// Mitsubishi GX Works2 project: plc0723   PLC: Q02/Q02H

// global labels: Global1
VAR_GLOBAL
  공급후 AT X0 : BOOL;
  공급전 AT X1 : BOOL;
  드릴상 AT X2 : BOOL;
  드릴하 AT X3 : BOOL;
  송출후 AT X4 : BOOL;
  송출전 AT X5 : BOOL;
  배출후 AT X6 : BOOL;
  배출전 AT X7 : BOOL;
  매거진 AT X8 : BOOL;
  비금속 AT X9 : BOOL;
  금속 AT X0A : BOOL;
  공급전솔 AT Y20 : BOOL;
  공급후솔 AT Y21 : BOOL;
  드릴온 AT Y22 : BOOL;
  송출전솔 AT Y23 : BOOL;
  송출후솔 AT Y24 : BOOL;
  배출전솔 AT Y25 : BOOL;
  배출후솔 AT Y26 : BOOL;
  컨베이어 AT Y27 : BOOL;
  가공드릴 AT Y28 : BOOL;
  적색 AT Y29 : BOOL;
  황색 AT Y2A : BOOL;
  녹색 AT Y2B : BOOL;
  pb1 AT X10 : BOOL;
  pb2 AT X11 : BOOL;
  pb3 AT X12 : BOOL;
  비상정지 AT X13 : BOOL;
  초기화 AT X14 : BOOL;
END_VAR

PROGRAM MAIN
VAR
  테스트동작 : BOOL;
  단일동작 : BOOL;
  연속동작 : BOOL;
  금속탐지 : BOOL;
  송출_전 : BOOL;
  공급_전 : BOOL;
  테스트타이머 : TIMER;
  공급_후 : BOOL;
  가공_하 : BOOL;
  배출_전 : BOOL;
  가공_상 : BOOL;
  배출_후 : BOOL;
  송출_후 : BOOL;
  테스트종료 : BOOL;
  황테 : BOOL;
  녹테 : BOOL;
  공급전진 : BOOL;
  물건없음 : TIMER;
  공급후진 : BOOL;
  타이머1 : TIMER;
  가공드릴온 : BOOL;
  드릴하강 : BOOL;
  타이머2 : TIMER;
  가공드릴오프 : BOOL;
  드릴상승 : BOOL;
  송출전진 : BOOL;
  송출후진 : BOOL;
  컨구동 : BOOL;
  금속판별 : BOOL;
  비금속판별 : BOOL;
  금속타이머 : TIMER;
  배출전진 : BOOL;
  배출후진 : BOOL;
  금종 : BOOL;
  비금속타이머 : TIMER;
  비종 : BOOL;
  동작종료 : BOOL;
  연속종료 : BOOL;
  공급전진2 : BOOL;
  녹색램프 : BOOL;
  황색램프 : BOOL;
  반전 : BOOL;
END_VAR
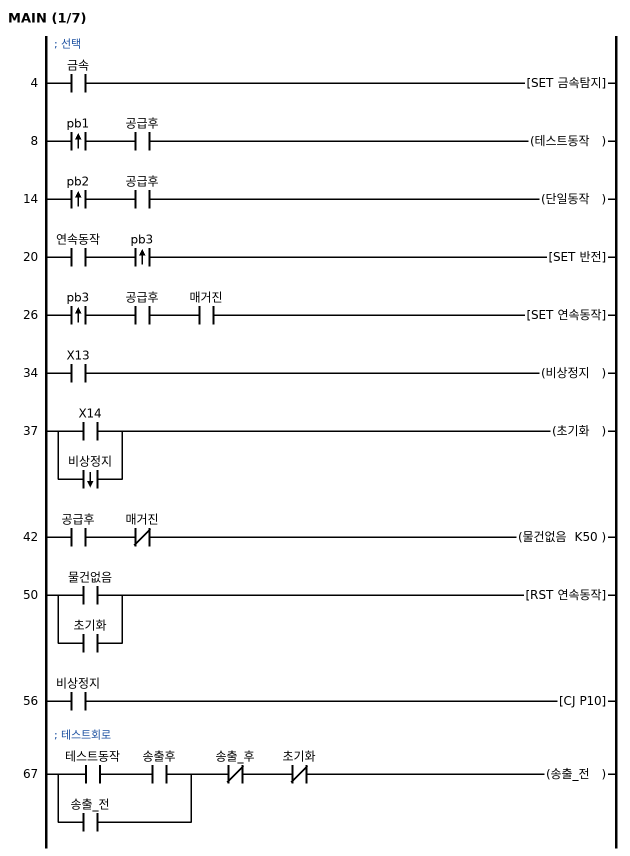
; 선택
4     LD      금속
      SET     금속탐지
8     LDP     pb1
      AND     공급후
      OUT     테스트동작
14    LDP     pb2
      AND     공급후
      OUT     단일동작
20    LD      연속동작
      ANDP    pb3
      SET     반전
26    LDP     pb3
      AND     공급후
      AND     매거진
      SET     연속동작
34    LD      X13
      OUT     비상정지
37    LD      X14
      ORF     비상정지
      OUT     초기화
42    LD      공급후
      ANI     매거진
      OUT     물건없음 K50
50    LD      물건없음
      OR      초기화
      RST     연속동작
56    LD      비상정지
      CJ      P10
; 테스트회로
67    LD      테스트동작
      AND     송출후
      OR      송출_전
      ANI     송출_후
      ANI     초기화
      OUT     송출_전
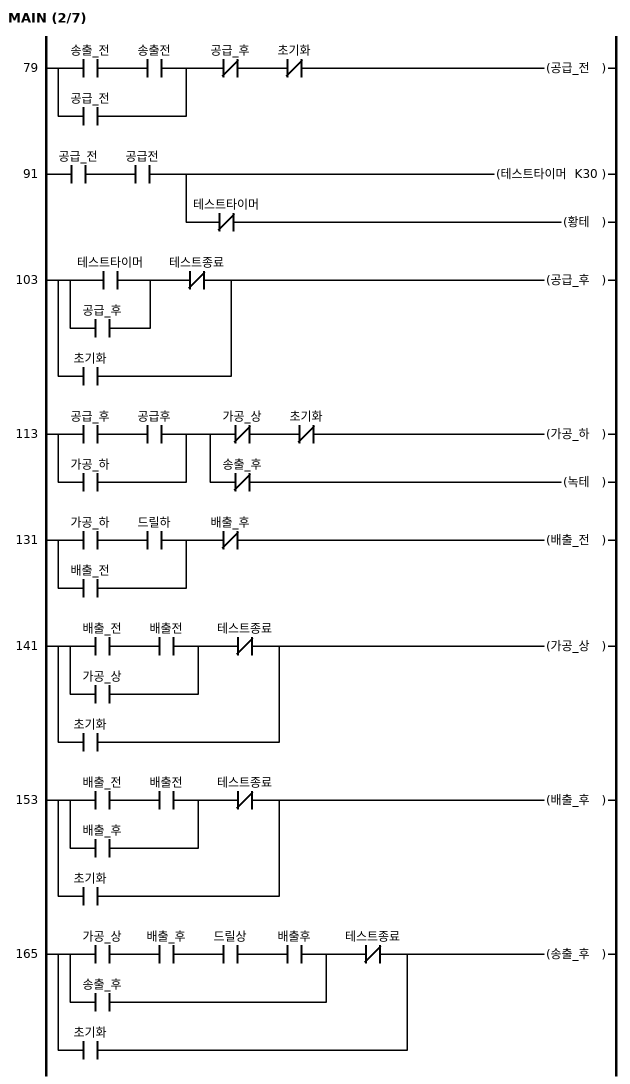
79    LD      송출_전
      AND     송출전
      OR      공급_전
      ANI     공급_후
      ANI     초기화
      OUT     공급_전
91    LD      공급_전
      AND     공급전
      OUT     테스트타이머 K30
      ANI     테스트타이머
      OUT     황테
103   LD      테스트타이머
      OR      공급_후
      ANI     테스트종료
      OR      초기화
      OUT     공급_후
113   LD      공급_후
      AND     공급후
      OR      가공_하
      MPS
      ANI     가공_상
      ANI     초기화
      OUT     가공_하
      MPP
      ANI     송출_후
      OUT     녹테
131   LD      가공_하
      AND     드릴하
      OR      배출_전
      ANI     배출_후
      OUT     배출_전
141   LD      배출_전
      AND     배출전
      OR      가공_상
      ANI     테스트종료
      OR      초기화
      OUT     가공_상
153   LD      배출_전
      AND     배출전
      OR      배출_후
      ANI     테스트종료
      OR      초기화
      OUT     배출_후
165   LD      가공_상
      AND     배출_후
      AND     드릴상
      AND     배출후
      OR      송출_후
      ANI     테스트종료
      OR      초기화
      OUT     송출_후
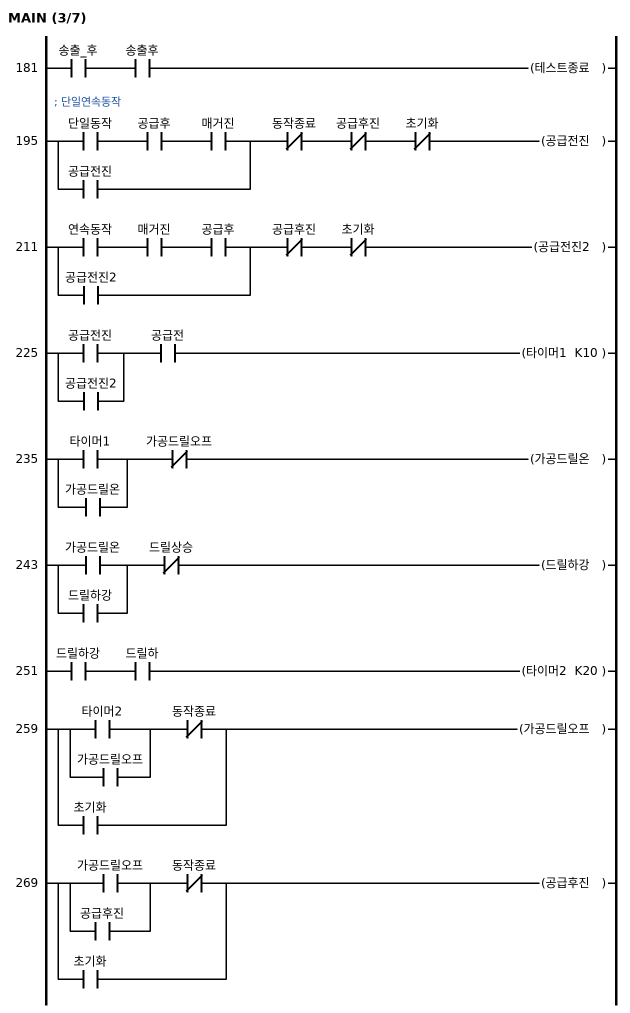
181   LD      송출_후
      AND     송출후
      OUT     테스트종료
; 단일연속동작
195   LD      단일동작
      AND     공급후
      AND     매거진
      OR      공급전진
      ANI     동작종료
      ANI     공급후진
      ANI     초기화
      OUT     공급전진
211   LD      연속동작
      AND     매거진
      AND     공급후
      OR      공급전진2
      ANI     공급후진
      ANI     초기화
      OUT     공급전진2
225   LD      공급전진
      OR      공급전진2
      AND     공급전
      OUT     타이머1 K10
235   LD      타이머1
      OR      가공드릴온
      ANI     가공드릴오프
      OUT     가공드릴온
243   LD      가공드릴온
      OR      드릴하강
      ANI     드릴상승
      OUT     드릴하강
251   LD      드릴하강
      AND     드릴하
      OUT     타이머2 K20
259   LD      타이머2
      OR      가공드릴오프
      ANI     동작종료
      OR      초기화
      OUT     가공드릴오프
269   LD      가공드릴오프
      OR      공급후진
      ANI     동작종료
      OR      초기화
      OUT     공급후진
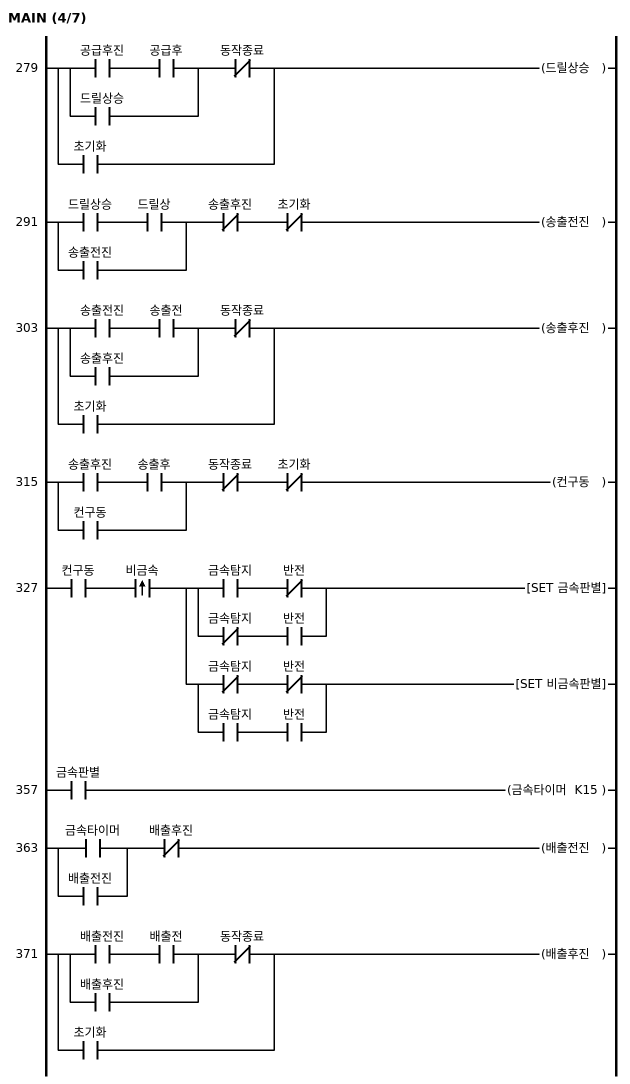
279   LD      공급후진
      AND     공급후
      OR      드릴상승
      ANI     동작종료
      OR      초기화
      OUT     드릴상승
291   LD      드릴상승
      AND     드릴상
      OR      송출전진
      ANI     송출후진
      ANI     초기화
      OUT     송출전진
303   LD      송출전진
      AND     송출전
      OR      송출후진
      ANI     동작종료
      OR      초기화
      OUT     송출후진
315   LD      송출후진
      AND     송출후
      OR      컨구동
      ANI     동작종료
      ANI     초기화
      OUT     컨구동
327   LD      컨구동
      ANDP    비금속
      MPS
      LD      금속탐지
      ANI     반전
      LDI     금속탐지
      AND     반전
      ORB
      ANB
      SET     금속판별
      MPP
      LDI     금속탐지
      ANI     반전
      LD      금속탐지
      AND     반전
      ORB
      ANB
      SET     비금속판별
357   LD      금속판별
      OUT     금속타이머 K15
363   LD      금속타이머
      OR      배출전진
      ANI     배출후진
      OUT     배출전진
371   LD      배출전진
      AND     배출전
      OR      배출후진
      ANI     동작종료
      OR      초기화
      OUT     배출후진
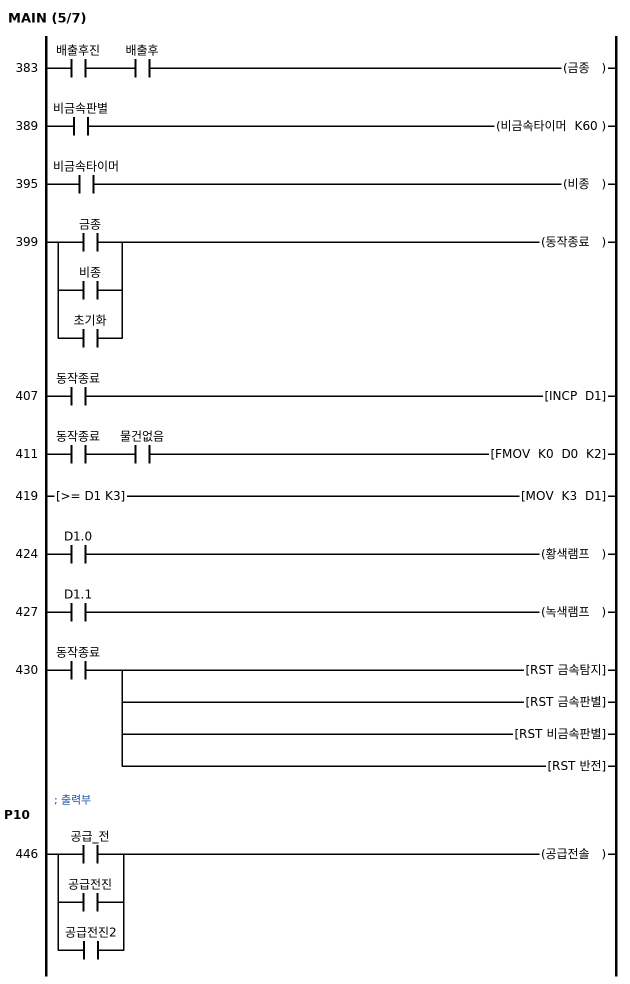
383   LD      배출후진
      AND     배출후
      OUT     금종
389   LD      비금속판별
      OUT     비금속타이머 K60
395   LD      비금속타이머
      OUT     비종
399   LD      금종
      OR      비종
      OR      초기화
      OUT     동작종료
407   LD      동작종료
      INCP    D1
411   LD      동작종료
      AND     물건없음
      FMOV    K0 D0 K2
419   LD>=    D1 K3
      MOV     K3 D1
424   LD      D1.0
      OUT     황색램프
427   LD      D1.1
      OUT     녹색램프
430   LD      동작종료
      RST     금속탐지
      RST     금속판별
      RST     비금속판별
      RST     반전
; 출력부
      P10
446   LD      공급_전
      OR      공급전진
      OR      공급전진2
      OUT     공급전솔
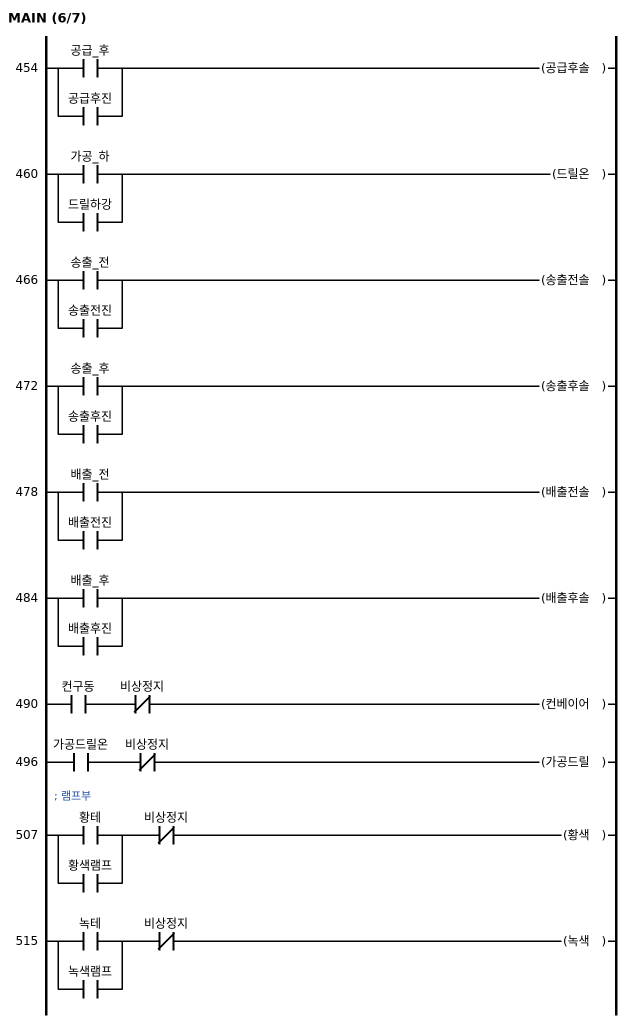
454   LD      공급_후
      OR      공급후진
      OUT     공급후솔
460   LD      가공_하
      OR      드릴하강
      OUT     드릴온
466   LD      송출_전
      OR      송출전진
      OUT     송출전솔
472   LD      송출_후
      OR      송출후진
      OUT     송출후솔
478   LD      배출_전
      OR      배출전진
      OUT     배출전솔
484   LD      배출_후
      OR      배출후진
      OUT     배출후솔
490   LD      컨구동
      ANI     비상정지
      OUT     컨베이어
496   LD      가공드릴온
      ANI     비상정지
      OUT     가공드릴
; 램프부
507   LD      황테
      OR      황색램프
      ANI     비상정지
      OUT     황색
515   LD      녹테
      OR      녹색램프
      ANI     비상정지
      OUT     녹색
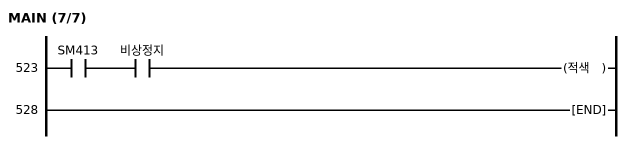
523   LD      SM413
      AND     비상정지
      OUT     적색
528   END
END_PROGRAM

PROGRAM test3
VAR
  테스트동작 : BOOL;
  단속동작 : BOOL;
  연속동작 : BOOL;
  공급_전 : BOOL;
  송출_전 : BOOL;
  송출_후 : BOOL;
  공급_후 : BOOL;
  테스트타이머 : TIMER;
  황테 : BOOL;
  테스트종료 : BOOL;
  배출_전 : BOOL;
  가공_하 : BOOL;
  배출_후 : BOOL;
  가공_상 : BOOL;
  녹색테스트 : BOOL;
  공급전진 : BOOL;
  공급후진 : BOOL;
  동작종료 : BOOL;
  가공드릴온 : BOOL;
  가공드릴오프 : BOOL;
  가공하강 : BOOL;
  가공상승 : BOOL;
  타이머1 : TIMER;
  타이머2 : TIMER;
  송출전진 : BOOL;
  송출후진 : BOOL;
  컨구동 : BOOL;
  금속탐지 : BOOL;
  비금속탐지 : BOOL;
  반전 : BOOL;
  금속판별 : BOOL;
  배출전진 : BOOL;
  비금속타이머 : TIMER;
  배출후진 : BOOL;
  비종 : BOOL;
  금속타이머 : TIMER;
  금종 : BOOL;
  공급전진2 : BOOL;
  물건없음 : TIMER;
  황색점등 : BOOL;
END_VAR
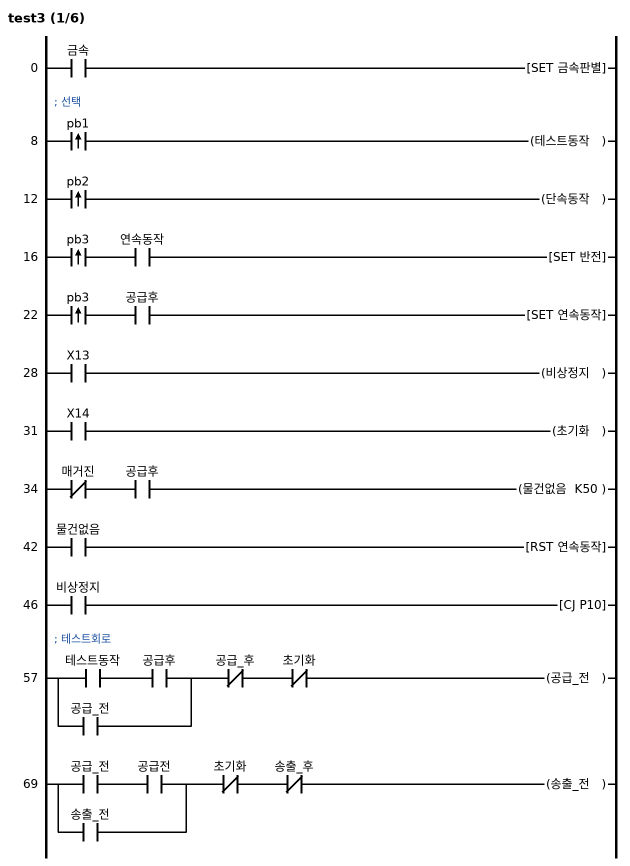
0     LD      금속
      SET     금속판별
; 선택
8     LDP     pb1
      OUT     테스트동작
12    LDP     pb2
      OUT     단속동작
16    LDP     pb3
      AND     연속동작
      SET     반전
22    LDP     pb3
      AND     공급후
      SET     연속동작
28    LD      X13
      OUT     비상정지
31    LD      X14
      OUT     초기화
34    LDI     매거진
      AND     공급후
      OUT     물건없음 K50
42    LD      물건없음
      RST     연속동작
46    LD      비상정지
      CJ      P10
; 테스트회로
57    LD      테스트동작
      AND     공급후
      OR      공급_전
      ANI     공급_후
      ANI     초기화
      OUT     공급_전
69    LD      공급_전
      AND     공급전
      OR      송출_전
      ANI     초기화
      ANI     송출_후
      OUT     송출_전
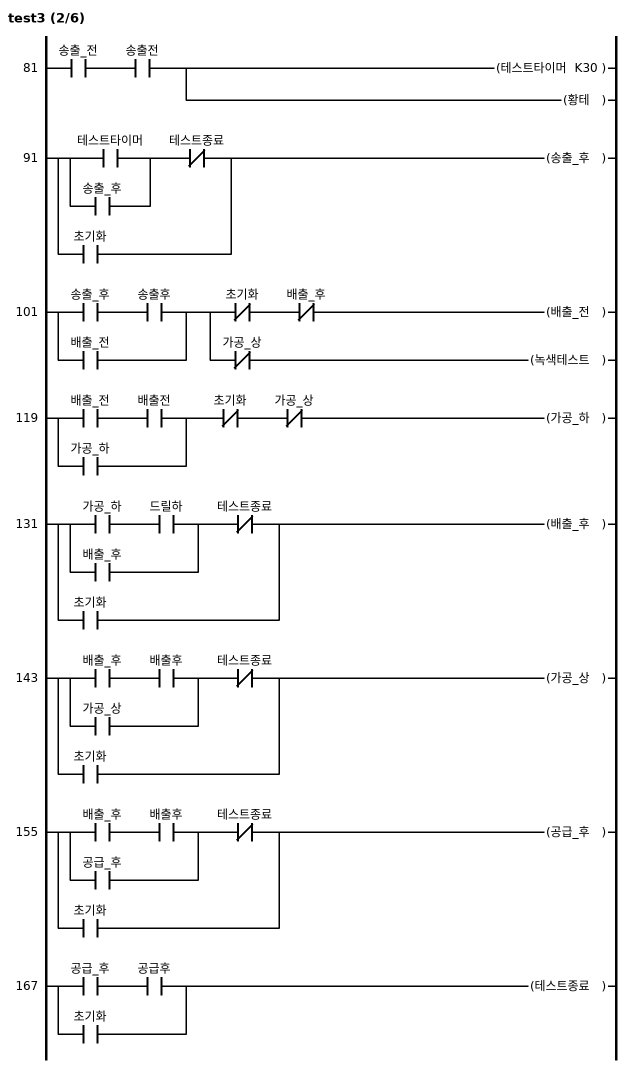
81    LD      송출_전
      AND     송출전
      OUT     테스트타이머 K30
      OUT     황테
91    LD      테스트타이머
      OR      송출_후
      ANI     테스트종료
      OR      초기화
      OUT     송출_후
101   LD      송출_후
      AND     송출후
      OR      배출_전
      MPS
      ANI     초기화
      ANI     배출_후
      OUT     배출_전
      MPP
      ANI     가공_상
      OUT     녹색테스트
119   LD      배출_전
      AND     배출전
      OR      가공_하
      ANI     초기화
      ANI     가공_상
      OUT     가공_하
131   LD      가공_하
      AND     드릴하
      OR      배출_후
      ANI     테스트종료
      OR      초기화
      OUT     배출_후
143   LD      배출_후
      AND     배출후
      OR      가공_상
      ANI     테스트종료
      OR      초기화
      OUT     가공_상
155   LD      배출_후
      AND     배출후
      OR      공급_후
      ANI     테스트종료
      OR      초기화
      OUT     공급_후
167   LD      공급_후
      AND     공급후
      OR      초기화
      OUT     테스트종료
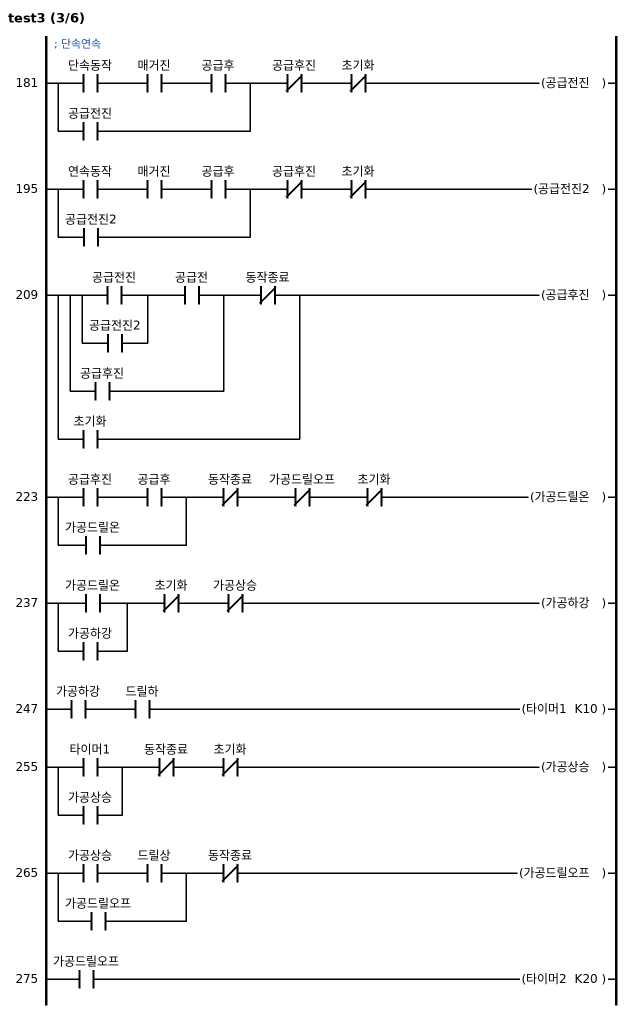
; 단속연속
181   LD      단속동작
      AND     매거진
      AND     공급후
      OR      공급전진
      ANI     공급후진
      ANI     초기화
      OUT     공급전진
195   LD      연속동작
      AND     매거진
      AND     공급후
      OR      공급전진2
      ANI     공급후진
      ANI     초기화
      OUT     공급전진2
209   LD      공급전진
      OR      공급전진2
      AND     공급전
      OR      공급후진
      ANI     동작종료
      OR      초기화
      OUT     공급후진
223   LD      공급후진
      AND     공급후
      OR      가공드릴온
      ANI     동작종료
      ANI     가공드릴오프
      ANI     초기화
      OUT     가공드릴온
237   LD      가공드릴온
      OR      가공하강
      ANI     초기화
      ANI     가공상승
      OUT     가공하강
247   LD      가공하강
      AND     드릴하
      OUT     타이머1 K10
255   LD      타이머1
      OR      가공상승
      ANI     동작종료
      ANI     초기화
      OUT     가공상승
265   LD      가공상승
      AND     드릴상
      OR      가공드릴오프
      ANI     동작종료
      OUT     가공드릴오프
275   LD      가공드릴오프
      OUT     타이머2 K20
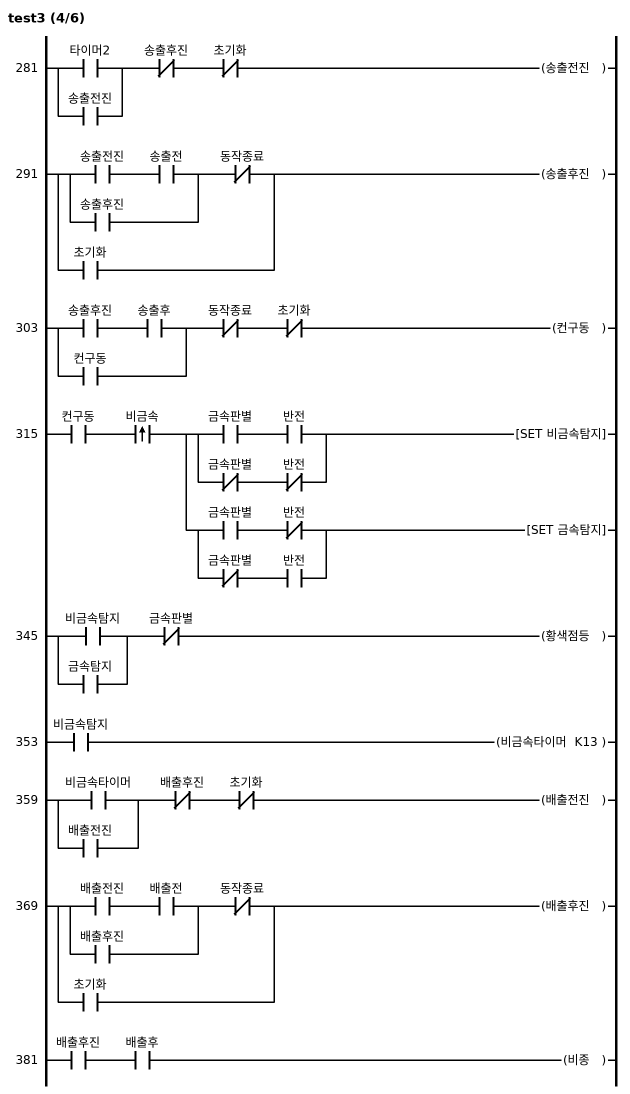
281   LD      타이머2
      OR      송출전진
      ANI     송출후진
      ANI     초기화
      OUT     송출전진
291   LD      송출전진
      AND     송출전
      OR      송출후진
      ANI     동작종료
      OR      초기화
      OUT     송출후진
303   LD      송출후진
      AND     송출후
      OR      컨구동
      ANI     동작종료
      ANI     초기화
      OUT     컨구동
315   LD      컨구동
      ANDP    비금속
      MPS
      LD      금속판별
      AND     반전
      LDI     금속판별
      ANI     반전
      ORB
      ANB
      SET     비금속탐지
      MPP
      LD      금속판별
      ANI     반전
      LDI     금속판별
      AND     반전
      ORB
      ANB
      SET     금속탐지
345   LD      비금속탐지
      OR      금속탐지
      ANI     금속판별
      OUT     황색점등
353   LD      비금속탐지
      OUT     비금속타이머 K13
359   LD      비금속타이머
      OR      배출전진
      ANI     배출후진
      ANI     초기화
      OUT     배출전진
369   LD      배출전진
      AND     배출전
      OR      배출후진
      ANI     동작종료
      OR      초기화
      OUT     배출후진
381   LD      배출후진
      AND     배출후
      OUT     비종
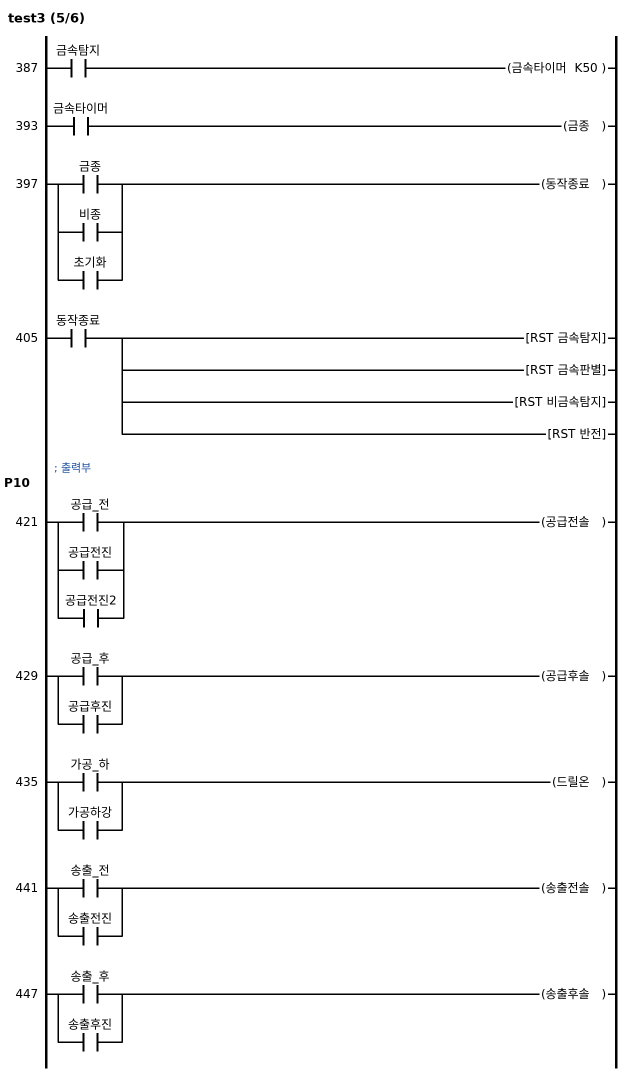
387   LD      금속탐지
      OUT     금속타이머 K50
393   LD      금속타이머
      OUT     금종
397   LD      금종
      OR      비종
      OR      초기화
      OUT     동작종료
405   LD      동작종료
      RST     금속탐지
      RST     금속판별
      RST     비금속탐지
      RST     반전
; 출력부
      P10
421   LD      공급_전
      OR      공급전진
      OR      공급전진2
      OUT     공급전솔
429   LD      공급_후
      OR      공급후진
      OUT     공급후솔
435   LD      가공_하
      OR      가공하강
      OUT     드릴온
441   LD      송출_전
      OR      송출전진
      OUT     송출전솔
447   LD      송출_후
      OR      송출후진
      OUT     송출후솔
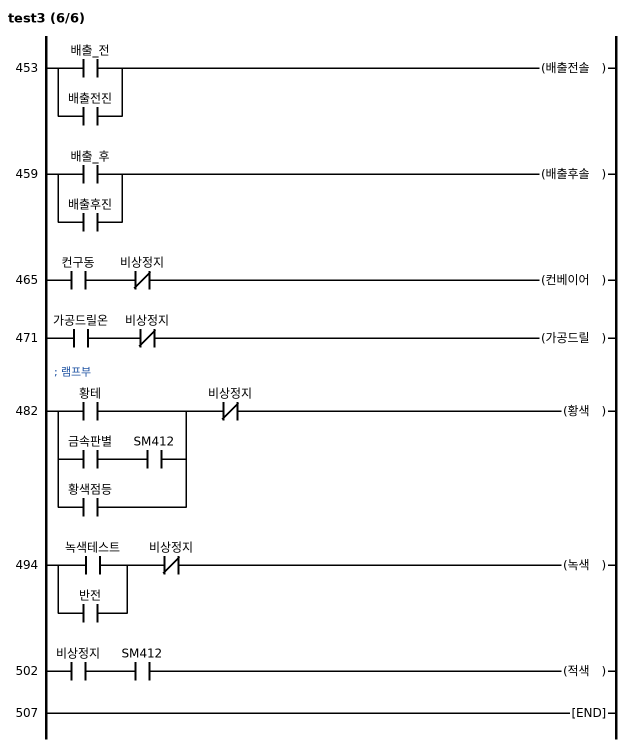
453   LD      배출_전
      OR      배출전진
      OUT     배출전솔
459   LD      배출_후
      OR      배출후진
      OUT     배출후솔
465   LD      컨구동
      ANI     비상정지
      OUT     컨베이어
471   LD      가공드릴온
      ANI     비상정지
      OUT     가공드릴
; 램프부
482   LD      황테
      LD      금속판별
      AND     SM412
      ORB
      OR      황색점등
      ANI     비상정지
      OUT     황색
494   LD      녹색테스트
      OR      반전
      ANI     비상정지
      OUT     녹색
502   LD      비상정지
      AND     SM412
      OUT     적색
507   END
END_PROGRAM

PROGRAM test4
VAR
  금속판별 : BOOL;
  테스트동작 : BOOL;
  단속동작 : BOOL;
  연속동작 : BOOL;
  공급_전 : BOOL;
  공급_후 : BOOL;
  테스트종료 : BOOL;
  가공_하 : BOOL;
  가공_상 : BOOL;
  송출_전 : BOOL;
  송출_후 : BOOL;
  테스트타이머 : TIMER;
  배출_전 : BOOL;
  배출_후 : BOOL;
  황테 : BOOL;
  녹테 : BOOL;
  공급전진 : BOOL;
  공급후진 : BOOL;
  공급전진2 : BOOL;
  동작종료 : BOOL;
  가공드릴온 : BOOL;
  가공드릴오프 : BOOL;
  타이머1 : TIMER;
  드릴하강 : BOOL;
  드릴상승 : BOOL;
  송출전진 : BOOL;
  송출후진 : BOOL;
  타이머2 : TIMER;
  컨구동 : BOOL;
  토글sw : BOOL;
  금속탐지 : BOOL;
  비금속탐지 : BOOL;
  금속타이머 : TIMER;
  금종 : BOOL;
  배출전진 : BOOL;
  배출후진 : BOOL;
  비금속타이머 : TIMER;
  비종 : BOOL;
  물건없음 : TIMER;
  초기화지연 : TIMER;
  초기화초기화 : BOOL;
  리셋 : BOOL;
  리셋타이머 : TIMER;
  돌아가 : BOOL;
END_VAR
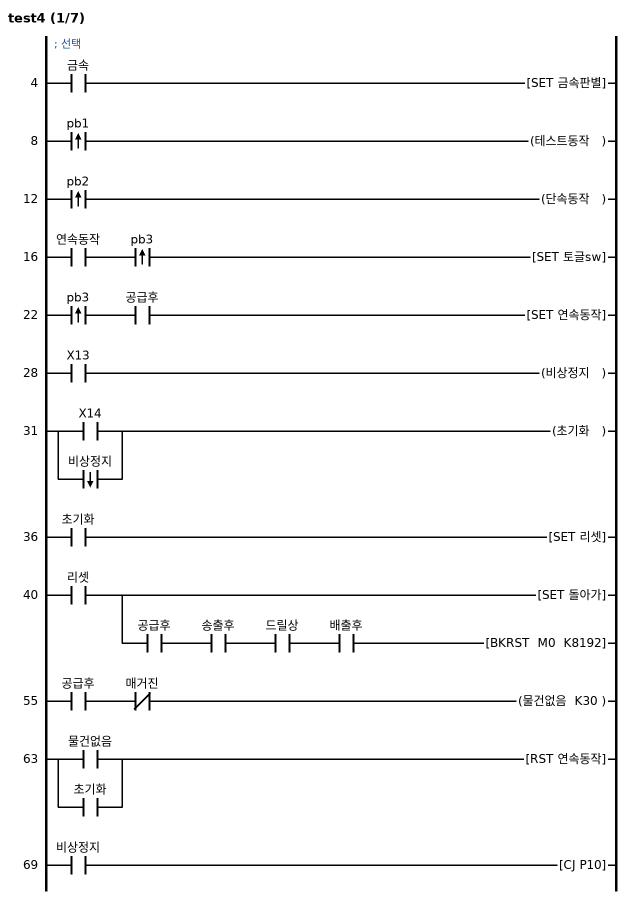
; 선택
4     LD      금속
      SET     금속판별
8     LDP     pb1
      OUT     테스트동작
12    LDP     pb2
      OUT     단속동작
16    LD      연속동작
      ANDP    pb3
      SET     토글sw
22    LDP     pb3
      AND     공급후
      SET     연속동작
28    LD      X13
      OUT     비상정지
31    LD      X14
      ORF     비상정지
      OUT     초기화
36    LD      초기화
      SET     리셋
40    LD      리셋
      SET     돌아가
      AND     공급후
      AND     송출후
      AND     드릴상
      AND     배출후
      BKRST   M0 K8192
55    LD      공급후
      ANI     매거진
      OUT     물건없음 K30
63    LD      물건없음
      OR      초기화
      RST     연속동작
69    LD      비상정지
      CJ      P10
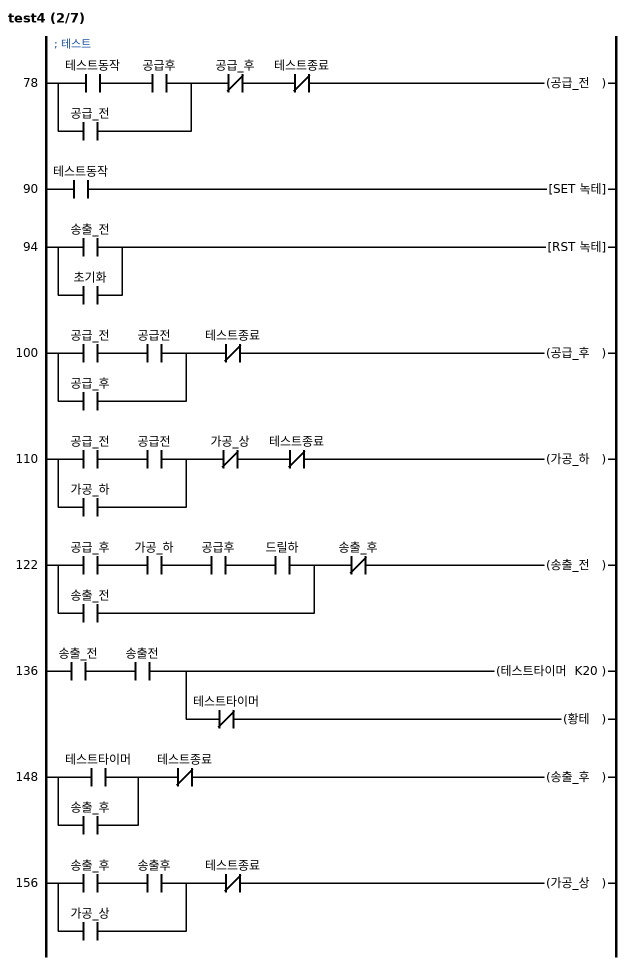
; 테스트
78    LD      테스트동작
      AND     공급후
      OR      공급_전
      ANI     공급_후
      ANI     테스트종료
      OUT     공급_전
90    LD      테스트동작
      SET     녹테
94    LD      송출_전
      OR      초기화
      RST     녹테
100   LD      공급_전
      AND     공급전
      OR      공급_후
      ANI     테스트종료
      OUT     공급_후
110   LD      공급_전
      AND     공급전
      OR      가공_하
      ANI     가공_상
      ANI     테스트종료
      OUT     가공_하
122   LD      공급_후
      AND     가공_하
      AND     공급후
      AND     드릴하
      OR      송출_전
      ANI     송출_후
      OUT     송출_전
136   LD      송출_전
      AND     송출전
      OUT     테스트타이머 K20
      ANI     테스트타이머
      OUT     황테
148   LD      테스트타이머
      OR      송출_후
      ANI     테스트종료
      OUT     송출_후
156   LD      송출_후
      AND     송출후
      OR      가공_상
      ANI     테스트종료
      OUT     가공_상
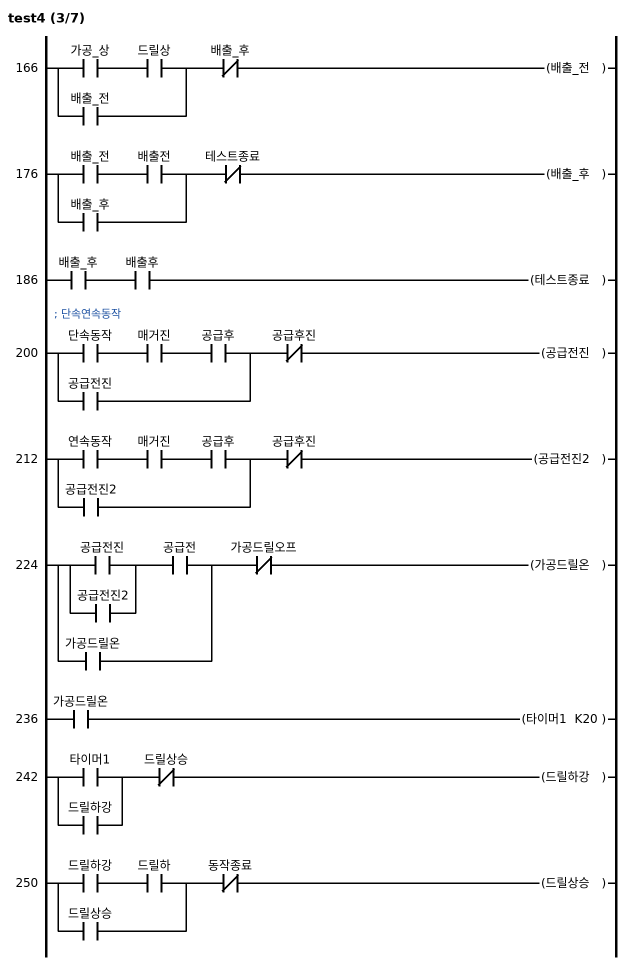
166   LD      가공_상
      AND     드릴상
      OR      배출_전
      ANI     배출_후
      OUT     배출_전
176   LD      배출_전
      AND     배출전
      OR      배출_후
      ANI     테스트종료
      OUT     배출_후
186   LD      배출_후
      AND     배출후
      OUT     테스트종료
; 단속연속동작
200   LD      단속동작
      AND     매거진
      AND     공급후
      OR      공급전진
      ANI     공급후진
      OUT     공급전진
212   LD      연속동작
      AND     매거진
      AND     공급후
      OR      공급전진2
      ANI     공급후진
      OUT     공급전진2
224   LD      공급전진
      OR      공급전진2
      AND     공급전
      OR      가공드릴온
      ANI     가공드릴오프
      OUT     가공드릴온
236   LD      가공드릴온
      OUT     타이머1 K20
242   LD      타이머1
      OR      드릴하강
      ANI     드릴상승
      OUT     드릴하강
250   LD      드릴하강
      AND     드릴하
      OR      드릴상승
      ANI     동작종료
      OUT     드릴상승
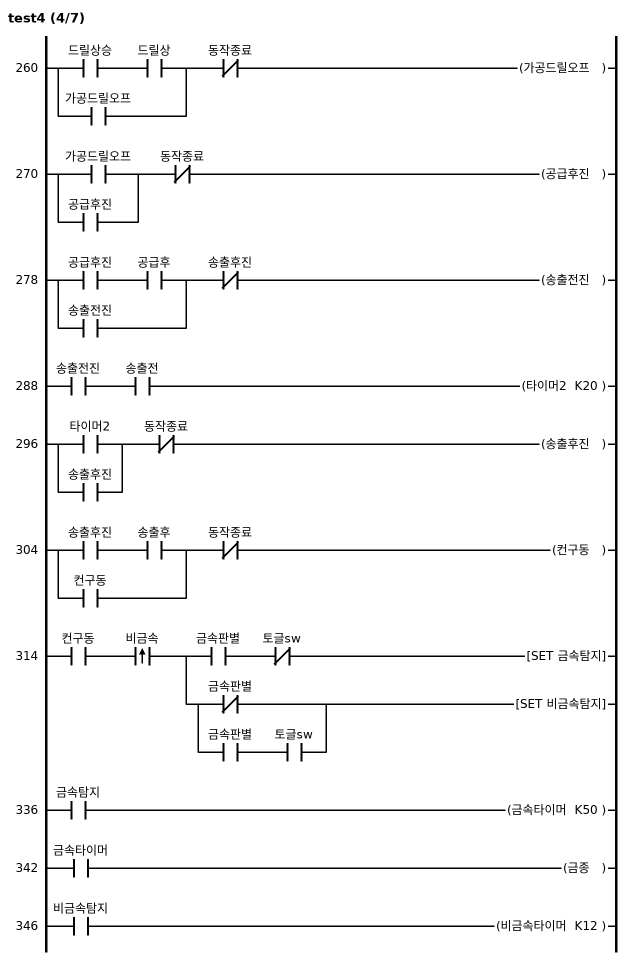
260   LD      드릴상승
      AND     드릴상
      OR      가공드릴오프
      ANI     동작종료
      OUT     가공드릴오프
270   LD      가공드릴오프
      OR      공급후진
      ANI     동작종료
      OUT     공급후진
278   LD      공급후진
      AND     공급후
      OR      송출전진
      ANI     송출후진
      OUT     송출전진
288   LD      송출전진
      AND     송출전
      OUT     타이머2 K20
296   LD      타이머2
      OR      송출후진
      ANI     동작종료
      OUT     송출후진
304   LD      송출후진
      AND     송출후
      OR      컨구동
      ANI     동작종료
      OUT     컨구동
314   LD      컨구동
      ANDP    비금속
      MPS
      AND     금속판별
      ANI     토글sw
      SET     금속탐지
      MPP
      LDI     금속판별
      LD      금속판별
      AND     토글sw
      ORB
      ANB
      SET     비금속탐지
336   LD      금속탐지
      OUT     금속타이머 K50
342   LD      금속타이머
      OUT     금종
346   LD      비금속탐지
      OUT     비금속타이머 K12
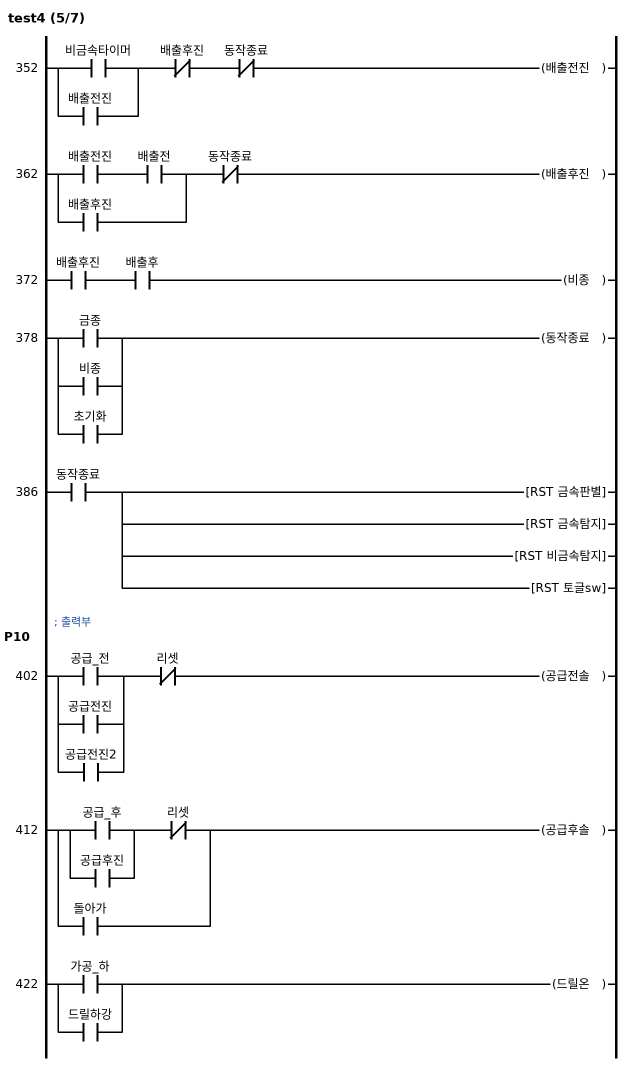
352   LD      비금속타이머
      OR      배출전진
      ANI     배출후진
      ANI     동작종료
      OUT     배출전진
362   LD      배출전진
      AND     배출전
      OR      배출후진
      ANI     동작종료
      OUT     배출후진
372   LD      배출후진
      AND     배출후
      OUT     비종
378   LD      금종
      OR      비종
      OR      초기화
      OUT     동작종료
386   LD      동작종료
      RST     금속판별
      RST     금속탐지
      RST     비금속탐지
      RST     토글sw
; 출력부
      P10
402   LD      공급_전
      OR      공급전진
      OR      공급전진2
      ANI     리셋
      OUT     공급전솔
412   LD      공급_후
      OR      공급후진
      ANI     리셋
      OR      돌아가
      OUT     공급후솔
422   LD      가공_하
      OR      드릴하강
      OUT     드릴온
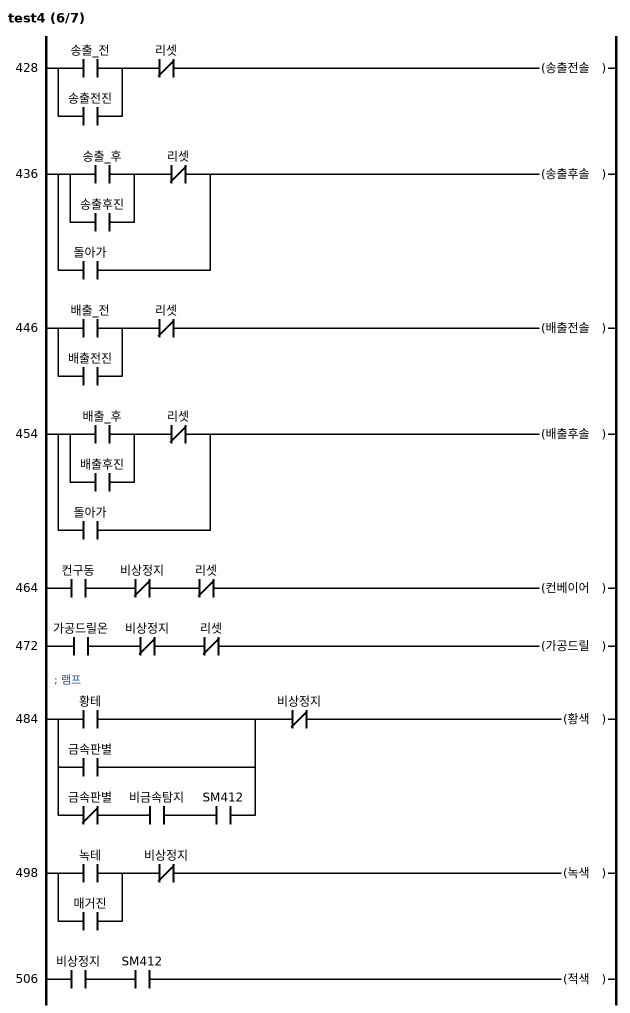
428   LD      송출_전
      OR      송출전진
      ANI     리셋
      OUT     송출전솔
436   LD      송출_후
      OR      송출후진
      ANI     리셋
      OR      돌아가
      OUT     송출후솔
446   LD      배출_전
      OR      배출전진
      ANI     리셋
      OUT     배출전솔
454   LD      배출_후
      OR      배출후진
      ANI     리셋
      OR      돌아가
      OUT     배출후솔
464   LD      컨구동
      ANI     비상정지
      ANI     리셋
      OUT     컨베이어
472   LD      가공드릴온
      ANI     비상정지
      ANI     리셋
      OUT     가공드릴
; 램프
484   LD      황테
      OR      금속판별
      LDI     금속판별
      AND     비금속탐지
      AND     SM412
      ORB
      ANI     비상정지
      OUT     황색
498   LD      녹테
      OR      매거진
      ANI     비상정지
      OUT     녹색
506   LD      비상정지
      AND     SM412
      OUT     적색
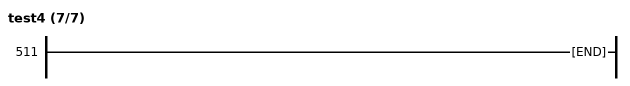
511   END
END_PROGRAM
